FUNCTION_BLOCK CAMERA (* Basic FB with empty ECC *)
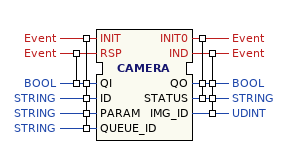
  EVENT_INPUT
    INIT WITH QI, PARAM, QUEUE_ID, ID;
    RSP WITH QI;
  END_EVENT
  EVENT_OUTPUT
    INIT0 WITH QO, STATUS;
    IND WITH QO, STATUS, IMG_ID;
  END_EVENT
  VAR_INPUT
    QI : BOOL;
    ID : STRING;
    PARAM : STRING;
    QUEUE_ID : STRING;
  END_VAR
  VAR_OUTPUT
    QO : BOOL;
    STATUS : STRING;
    IMG_ID : UDINT;
  END_VAR
END_FUNCTION_BLOCK
